{attribute 'GeneratedUsingTerminal: EL3111-0000-0016'}
{attribute addProperty BoxType "EL3111-0000-0016"}
{attribute addProperty Description "EL3111 1Ch. Ana. Input 0-20mA, Diff."}
{attribute addProperty Physics "KK"}
{attribute addProperty Id "AI_StandardAT %I*AI_Standard_A8DF64E310WcStateAT %I*WcState_9091E0EB2InfoDataAT %I*InfoData_32EB74EA10"}
{attribute addProperty CRC "2916756744"}
{attribute addProperty Size "22"}
TYPE EL3111_ADDA2D08 EXTENDS EtcSlaveTerminalBase_947E5A46 :
STRUCT
	{attribute addProperty Name "AI_Standard"}
	AI_Standard : AI_Standard_A8DF64E3;
	{attribute addProperty Name "WcState"}
	WcState : WcState_9091E0EB;
	{attribute addProperty Name "InfoData"}
	InfoData : InfoData_32EB74EA;
END_STRUCT
END_TYPE

(* stored: Version 1.2.0.0, ProductVersion 3.1.4024.9
   DUT EL3111_ADDA2D08: Id {1357cf30-0b0b-48da-ad45-c531e39dc9d5} *)
